FUNCTION_BLOCK TcoAbbRoboticsTest EXTENDS TcoAbbRobotics.TcoIrc5_v_1_x_x
VAR
    _serviceModeCount : ULINT;
    _serviceModeOverride : LREAL;
END_VAR
VAR
END_VAR

//SUPER^(	inEnable 			:=	inEnable,
//		inEnablePositive	:=	inEnablePositive,
//		inEnableNegative	:=	inEnableNegative,
//		inCalibrationCam	:=	inCalibrationCam,
//		inoAxisRef			:=	inoAxisRef);
//

END_FUNCTION_BLOCK

(* stored: Version 1.1.0.1, ProductVersion 3.1.4024.12
   POU TcoAbbRoboticsTest: Id {a0b286ed-8bfb-074f-019a-9e32adef0be7}, SpecialFunc None *)
